# EPICS autosave request: iocBoot/iocRontec/auto_settings.req
file "mca_settings.req",          P=$(P), M=mca1
file "RontecXFlash_settings.req", P=$(P), R=Rontec1
